FUNCTION_BLOCK CentralServerClient (* Client Function Block Type for Central Server ME Algorithm *)
  (* Standard: 61499-2 *)
  (* Version 0.2, 2003-12-04, JHC, Rockwell Automation, Renamed for better indexing. *)
  (* Version 0.1, 2002-11-05, JHC, Rockwell Automation, Corrected missing ST element in Algorithm REQ. *)
  (* Version 0.0, 2000-05-30, JHC, Rockwell Automation *)
  (* Compiler header: package fb.rt.cs725; *)
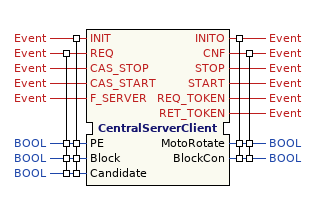
  EVENT_INPUT
    INIT WITH PE, Block, Candidate; (* Initialization Request *)
    REQ WITH PE, Block, Candidate; (* Normal Execution Request *)
    CAS_STOP;
    CAS_START;
    F_SERVER;
  END_EVENT
  EVENT_OUTPUT
    INITO WITH MotoRotate, BlockCon; (* Initialization Confirm *)
    CNF WITH MotoRotate, BlockCon; (* Execution Confirmation *)
    STOP;
    START;
    REQ_TOKEN;
    RET_TOKEN;
  END_EVENT
  VAR_INPUT
    PE : BOOL; (* Input event qualifier *)
    Block : BOOL;
    Candidate : BOOL;
  END_VAR
  VAR_OUTPUT
    MotoRotate : BOOL; (* Output event qualifier *)
    BlockCon : BOOL;
  END_VAR
  VAR
    lastPE : BOOL := 1;
    lastBlock : BOOL := 0;
  END_VAR
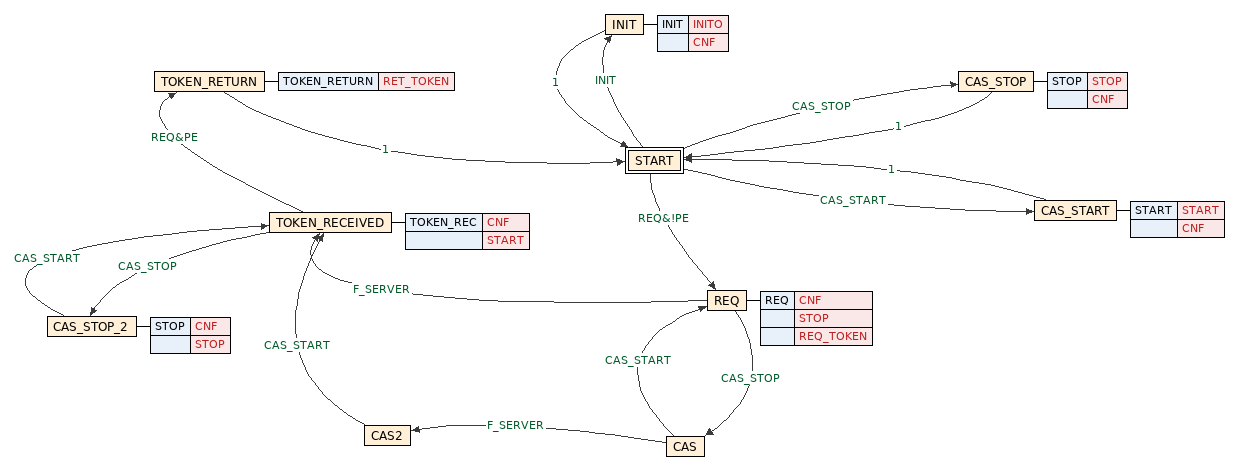
  EC_STATES
    START; (* Initial State *)
    INIT : INIT -> INITO, -> CNF; (* Initialization *)
    REQ : REQ -> CNF, -> STOP, -> REQ_TOKEN; (* Normal execution *)
    CAS_START : START -> START, -> CNF;
    CAS_STOP : STOP -> STOP, -> CNF;
    TOKEN_RECEIVED : TOKEN_REC -> CNF, -> START;
    TOKEN_RETURN : TOKEN_RETURN -> RET_TOKEN;
    CAS_STOP_2 : STOP -> CNF, -> STOP;
    CAS;
    CAS2;
  END_STATES
  EC_TRANSITIONS
    START TO INIT := INIT;
    INIT TO START := 1;
    START TO REQ := REQ&!PE;
    START TO CAS_START := CAS_START;
    CAS_START TO START := 1;
    START TO CAS_STOP := CAS_STOP;
    CAS_STOP TO START := 1;
    REQ TO TOKEN_RECEIVED := F_SERVER;
    TOKEN_RECEIVED TO TOKEN_RETURN := REQ&PE;
    TOKEN_RETURN TO START := 1;
    TOKEN_RECEIVED TO CAS_STOP_2 := CAS_STOP;
    CAS_STOP_2 TO TOKEN_RECEIVED := CAS_START;
    REQ TO CAS := CAS_STOP;
    CAS TO CAS2 := F_SERVER;
    CAS TO REQ := CAS_START;
    CAS2 TO TOKEN_RECEIVED := CAS_START;
  END_TRANSITIONS
  ALGORITHM INIT IN ST: (* Initialization algorithm *)
MotoRotate := TRUE;
Block := FALSE;
  END_ALGORITHM
  ALGORITHM REQ IN Java: (* Normally executed algorithm *)
System.out.println("----------------");
System.out.println("BAG DETECTED BY IN CS1");
System.out.println("----------------");
MotoRotate.value=false;
  END_ALGORITHM
  ALGORITHM START IN Java:
MotoRotate.value=true;
  END_ALGORITHM
  ALGORITHM STOP IN Java:
MotoRotate.value=false;
  END_ALGORITHM
  ALGORITHM TOKEN_REC IN Java:
MotoRotate.value=true;
System.out.println("----------------");
System.out.println("TOKEN RECEIVED IN CS 1") ;
System.out.println("----------------");
  END_ALGORITHM
  ALGORITHM TOKEN_RETURN IN Java:
System.out.println("----------------");
System.out.println("TOKEN IS BEING RETURNED in CS 1");
System.out.println("----------------");
  END_ALGORITHM
END_FUNCTION_BLOCK
